FUNCTION_BLOCK SimpleRelay EXTENDS SM_SimpleRelay
VAR_INPUT
END_VAR
VAR_OUTPUT
END_VAR
VAR
    testVar : INT;
END_VAR

_update();
_switching();
_update();

METHOD _update
VAR_INPUT
END_VAR
SUPER^();

IF digitalOutput THEN
    actualStatus := 'Enabled';
ELSE
    actualStatus := 'Disabled';
END_IF
END_METHOD

METHOD _switching
VAR_INPUT
END_VAR
IF processes.setEnabled.isBusy() THEN
    
    digitalOutput := processes.setEnabled.get.enabled;

    processes.setEnabled.setGood();
    processes.setEnabled.setFinished();
    
END_IF
END_METHOD

END_FUNCTION_BLOCK

(* stored: Version 1.1.0.1, ProductVersion 3.1.4018.2
   POU SimpleRelay: Id {813bf4c8-d588-42a3-94d7-69ffc697bd98}, SpecialFunc None
   Method _update: Id {79909a61-c6dd-4de5-a106-e4b2e9a97ada}
   Method _switching: Id {ae4ee04b-e071-4667-97f1-f2ff29622115} *)
